TYPE ST_InfoDataGroup :
STRUCT
	usiMapState: USINT;
	usiMapDiag: USINT;
END_STRUCT
END_TYPE

(* stored: Version 1.1.0.1
   DUT ST_InfoDataGroup: Id {ac28ab7e-1c6e-4c96-aa10-5ecb381f8a29} *)
